(* Verfiy that the state of the devices in the transport tube specified are in the expected state *)
FUNCTION F_VerifyTransportTubeStatuses : BOOL
VAR_INPUT
	stExpStatus : ST_TransportTubeStatuses;
	stStatusOp : ST_TransportTubeOps;
	eTransportTube : E_TransportTube;
	bEnforce : BOOL;
END_VAR
VAR
	stStatus : ST_TransportTubeStatuses;
END_VAR

stStatus := F_GetTransportTubeStatuses(eTransportTube);

IF bEnforce THEN
	// Try setting system states to the expected states
	F_SetTransportTubeStatuses(eTransportTube := eTransportTube, stExpStatus := stExpStatus, stStatusOp := stStatusOp);
END_IF

F_VerifyTransportTubeStatuses := (stExpStatus.bIonPumpOn = stStatus.bIonPumpOn OR stStatusOp.bIonPumpIgnore)
	AND (stExpStatus.bGateValveOpen = stStatus.bGateValveOpen OR stStatusOp.bGateValveIgnore)
	AND F_CompareGauge(eCompOp := stStatusOp.ePiraniOp, 
		fReading := stStatus.fPiraniGaugeVal, 
		eState := stStatus.ePiraniGaugeState, 
		fExpReading := stExpStatus.fPiraniGaugeVal, 
		eExpState := stExpStatus.ePiraniGaugeState)
	AND F_CompareGauge(eCompOp := stStatusOp.eColdCathodeOp, 
		fReading := stStatus.fColdCathodeVal, 
		eState := stStatus.eColdCathodeState,
		fExpReading := stExpStatus.fColdCathodeVal,
		eExpState := stExpStatus.eColdCathodeState);

END_FUNCTION

(* stored: Version 1.1.0.1, ProductVersion 3.1.4024.0
   POU F_VerifyTransportTubeStatuses: Id {1541c929-edac-0f9d-296a-dec165f0fa68}, SpecialFunc None *)
